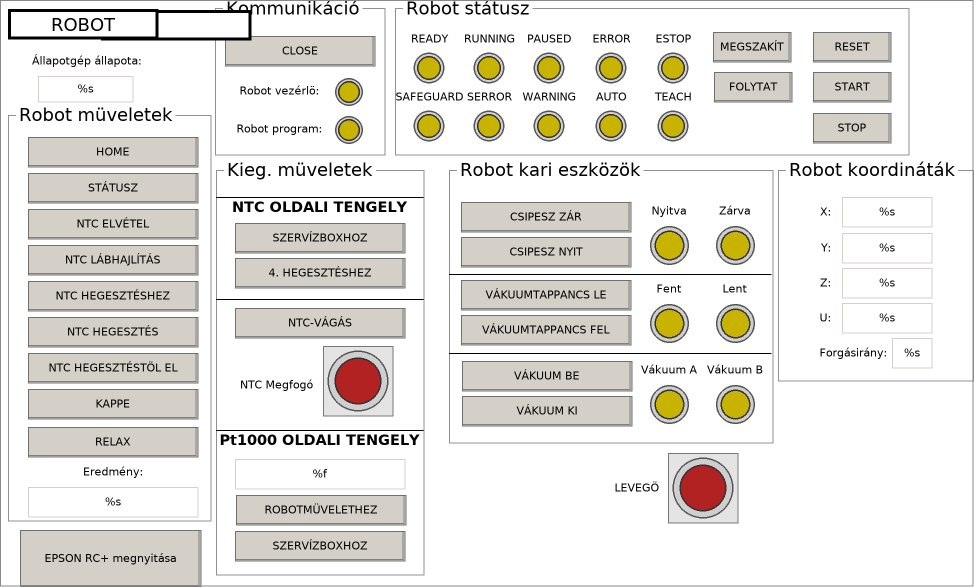
VISUALIZATION Robot  // 974x587
    GroupBox (215,0 170x155), "Kommunikáció"
        Button (10,36 150x30), "OPEN", invisible if: RobotProcess.iState>0, input disabled if: RobotProcess.iState>0
            OnMouseClick: execute { RobotProcess.iState:=1; }
        Button (10,36 150x30), "CLOSE", invisible if: RobotProcess.iState=0, input disabled if: RobotProcess.iState=0
            OnMouseClick: execute { RobotProcess.iState:=200; }
        Lamp1 (116,76 36x32), variable: ROBOTREMOTE.bRobotCommOpen, style: Lamp-Lamp1-Yellow
        Label (23,81 84x20), "Robot vezérlö:"
        Label (9,119 101x20), "Robot program:"
        Lamp1 (116,114 36x32), variable: ROBOTCOMMAND.bRobotCommOpen, style: Lamp-Lamp1-Yellow
    GroupBox (395,0 514x155), "Robot státusz", invisible if: RobotProcess.iState=0, input disabled if: RobotProcess.iState=0
        Lamp1 (16,50 36x36), variable: RobotProcess.baStatus[10], invisible if: ROBOTREMOTE.bRobotCommOpen=FALSE, style: Lamp-Lamp1-Yellow
        Label (6,24 57x30), "READY", invisible if: ROBOTREMOTE.bRobotCommOpen=FALSE
        Lamp1 (76,50 36x36), variable: RobotProcess.baStatus[9], invisible if: ROBOTREMOTE.bRobotCommOpen=FALSE, style: Lamp-Lamp1-Yellow
        Label (66,24 57x30), "RUNNING", invisible if: ROBOTREMOTE.bRobotCommOpen=FALSE
        Lamp1 (136,50 36x36), variable: RobotProcess.baStatus[8], invisible if: ROBOTREMOTE.bRobotCommOpen=FALSE, style: Lamp-Lamp1-Yellow
        Label (126,24 57x30), "PAUSED", invisible if: ROBOTREMOTE.bRobotCommOpen=FALSE
        Lamp1 (198,50 36x36), variable: RobotProcess.baStatus[7], invisible if: ROBOTREMOTE.bRobotCommOpen=FALSE, style: Lamp-Lamp1-Yellow
        Label (188,24 57x30), "ERROR", invisible if: ROBOTREMOTE.bRobotCommOpen=FALSE
        Lamp1 (260,50 36x36), variable: RobotProcess.baStatus[6], invisible if: ROBOTREMOTE.bRobotCommOpen=FALSE, style: Lamp-Lamp1-Yellow
        Label (250,24 57x30), "ESTOP", invisible if: ROBOTREMOTE.bRobotCommOpen=FALSE
        Lamp1 (16,108 36x36), variable: RobotProcess.baStatus[5], invisible if: ROBOTREMOTE.bRobotCommOpen=FALSE, style: Lamp-Lamp1-Yellow
        Label (6,82 57x30), "SAFEGUARD", invisible if: ROBOTREMOTE.bRobotCommOpen=FALSE
        Lamp1 (76,108 36x36), variable: RobotProcess.baStatus[4], invisible if: ROBOTREMOTE.bRobotCommOpen=FALSE, style: Lamp-Lamp1-Yellow
        Label (66,82 57x30), "SERROR", invisible if: ROBOTREMOTE.bRobotCommOpen=FALSE
        Lamp1 (136,108 36x36), variable: RobotProcess.baStatus[3], invisible if: ROBOTREMOTE.bRobotCommOpen=FALSE, style: Lamp-Lamp1-Yellow
        Label (126,82 57x30), "WARNING", invisible if: ROBOTREMOTE.bRobotCommOpen=FALSE
        Lamp1 (198,108 36x36), variable: RobotProcess.baStatus[2], invisible if: ROBOTREMOTE.bRobotCommOpen=FALSE, style: Lamp-Lamp1-Yellow
        Label (188,82 57x30), "AUTO", invisible if: ROBOTREMOTE.bRobotCommOpen=FALSE
        Lamp1 (260,108 36x36), variable: RobotProcess.baStatus[1], invisible if: ROBOTREMOTE.bRobotCommOpen=FALSE, style: Lamp-Lamp1-Yellow
        Label (250,82 57x30), "TEACH", invisible if: ROBOTREMOTE.bRobotCommOpen=FALSE
        RoundedRectangle (-294,10 150x30)
        Button (318,32 78x30), "MEGSZAKÍT"
            OnMouseClick: execute { ROBOTREMOTE.sRobotCommand := 'Pause'; ROBOTREMOTE.bRobotCommandSend := TRUE; }
        Button (319,72 78x30), "FOLYTAT"
            OnMouseClick: execute { ROBOTREMOTE.sRobotCommand := 'Continue'; ROBOTREMOTE.bRobotCommandSend := TRUE; }
        Button (418,32 78x30), "RESET"
            OnMouseClick: execute { ROBOTREMOTE.sRobotCommand := 'Reset'; ROBOTREMOTE.bRobotCommandSend := TRUE; }
        Button (418,72 78x30), "START"
            OnMouseClick: execute {
                ROBOTREMOTE.sRobotCommand := 'Start';
                ROBOTREMOTE.sRobotCommandParam1 := '0';
                ROBOTREMOTE.bRobotCommandSend := TRUE;
            }
        Button (418,113 78x30), "STOP"
            OnMouseClick: execute { ROBOTREMOTE.sRobotCommand := 'Stop'; ROBOTREMOTE.bRobotCommandSend := TRUE; }
    GroupBox (8,107 203x414), "Robot müveletek", invisible if: RobotProcess.iState=0, input disabled if: RobotProcess.iState=0
        Button (20,102 170x30), "NTC ELVÉTEL", invisible if: RobotProcess.iState=0, input disabled if: RobotProcess.iState=0
            OnMouseClick: execute { RobotProcess.s_InRobotTCPCommand := 'NTCHEZ'; }
        Button (20,174 170x30), "NTC HEGESZTÉSHEZ", invisible if: RobotProcess.iState=0, input disabled if: RobotProcess.iState=0
            OnMouseClick: execute { RobotProcess.s_InRobotTCPCommand := 'NTCHEG'; }
        Button (20,246 170x30), "NTC HEGESZTÉSTÖL EL", invisible if: RobotProcess.iState=0, input disabled if: RobotProcess.iState=0
            OnMouseClick: execute { RobotProcess.s_InRobotTCPCommand := 'NTCHEGTOL'; }
        Button (20,282 170x30), "KAPPE", invisible if: RobotProcess.iState=0, input disabled if: RobotProcess.iState=0
            OnMouseClick: execute { RobotProcess.s_InRobotTCPCommand := 'KAPPE'; }
        Button (20,320 170x30), "RELAX", invisible if: RobotProcess.iState=0, input disabled if: RobotProcess.iState=0
            OnMouseClick: execute { RobotProcess.s_InRobotTCPCommand := 'RELAX'; }
        Button (20,30 170x30), "HOME", invisible if: RobotProcess.iState=0, input disabled if: RobotProcess.iState=0
            OnMouseClick: execute { RobotProcess.s_InRobotTCPCommand := 'HOME'; }
        Textfield (20,380 170x30), "%s", text variable: ROBOTCOMMAND.sRobotResult, input disabled if: TRUE
        Label (60,350 90x30), "Eredmény:"
        Button (20,138 170x30), "NTC LÁBHAJLÍTÁS", invisible if: RobotProcess.iState=0, input disabled if: RobotProcess.iState=0
            OnMouseClick: execute { RobotProcess.s_InRobotTCPCommand := 'NTCLAB'; }
        Button (20,66 170x30), "STÁTUSZ", invisible if: RobotProcess.iState=0, input disabled if: RobotProcess.iState=0
            OnMouseClick: execute { RobotProcess.s_InRobotTCPCommand := 'STATUSZ'; }
        Button (20,210 170x30), "NTC HEGESZTÉS", invisible if: RobotProcess.iState=0, input disabled if: RobotProcess.iState=0
            OnMouseClick: execute {
                IF ROBOTCOMMAND.sRobotResult='NTCHEG' THEN
                	RobotProcess.s_InRobotTCPCommand := 'NTCHEG2';
                END_IF
            }
    Textfield (38,76 95x26), "%s", text variable: RobotProcess.iState, input disabled if: TRUE
    GroupBox (216,162 208x413), "Kieg. müveletek", invisible if: RobotProcess.iState=0, input disabled if: RobotProcess.iState=0
        Button (19,146 170x30), "NTC-VÁGÁS", input disabled if: NTCProcess.s_InCommand <> ''
            OnMouseUp: execute {
                IF NTCProcess.s_InCommand = '' THEN
                	NTCProcess.s_InCommand:='VAGAS';
                END_IF
            }
        Button (19,96 170x30), "4. HEGESZTÉSHEZ"
            OnMouseUp: execute { JOZSITENGELY.lrJozsiPosition:=GVL.lrHegesztoPosition4; JOZSITENGELY.sJozsiAxisCommand:='MOVE'; }
        PushSwitch (107,184 70x70), variable: NTCProcess.bMegfogo, behaviour: TOGGLE, style: Switch-PushSwitch-Red
        Label (17,213 87x20), "NTC Megfogó"
        Textfield (19,297 170x30), "%f", text variable: GVL.lrRobotKappePosition
            OnMouseClick: write the text variable via VisuDialogs.Numpad, min -10000, max -1
        Button (19,61 170x30), "SZERVÍZBOXHOZ"
            OnMouseUp: execute { JOZSITENGELY.lrJozsiPosition:=GVL.lrNTCSzervizbox; JOZSITENGELY.sJozsiAxisCommand:='MOVE'; }
        Button (19,369 170x30), "SZERVÍZBOXHOZ"
            OnMouseUp: execute { PISTITENGELY.lrPistiPosition:=GVL.lrPtSzervizbox; PISTITENGELY.sPistiAxisCommand:='MOVE'; }
        Line (0,268) (207,268), "Pt1000 OLDALI TENGELY"
        Line (0,35) (207,35), "NTC OLDALI TENGELY"
        Line (0,137) (207,137)
        Button (20,333 170x30), "ROBOTMÜVELETHEZ"
            OnMouseUp: execute { PISTITENGELY.lrPistiPosition:=GVL.lrRobotKappePosition; PISTITENGELY.sPistiAxisCommand:='MOVE'; }
    Label (27,46 120x30), "Állapotgép állapota:"
    RoundedRectangle (8,9 150x30)
    Label (8,10 150x30), "ROBOT"
    GroupBox (449,162 324x281), "Robot kari eszközök", invisible if: RobotProcess.iState=0, input disabled if: RobotProcess.iState=0
        Button (12,40 170x30), "CSIPESZ ZÁR", invisible if: RobotProcess.iState=0, input disabled if: RobotProcess.iState=0
            OnMouseClick: execute { RobotProcess.s_InRobotTCPCommand := 'CSIPESZ_ZAR'; }
        Button (12,75 170x30), "CSIPESZ NYIT", invisible if: RobotProcess.iState=0, input disabled if: RobotProcess.iState=0
            OnMouseClick: execute { RobotProcess.s_InRobotTCPCommand := 'CSIPESZ_NYIT'; }
        Group (12,118 170x65)
            Button (0,0 170x30), "VÁKUUMTAPPANCS LE", invisible if: RobotProcess.iState=0, input disabled if: RobotProcess.iState=0
                OnMouseClick: execute { RobotProcess.s_InRobotTCPCommand := 'SZIPPANTO_LE'; }
            Button (0,35 170x30), "VÁKUUMTAPPANCS FEL", invisible if: RobotProcess.iState=0, input disabled if: RobotProcess.iState=0
                OnMouseClick: execute { RobotProcess.s_InRobotTCPCommand := 'SZIPPANTO_FEL'; }
        Group (13,199 170x65)
            Button (0,35 170x30), "VÁKUUM KI", invisible if: RobotProcess.iState=0, input disabled if: RobotProcess.iState=0
                OnMouseClick: execute { RobotProcess.s_InRobotTCPCommand := 'VAKUUM_KI'; }
            Button (0,0 170x30), "VÁKUUM BE", invisible if: RobotProcess.iState=0, input disabled if: RobotProcess.iState=0
                OnMouseClick: execute { RobotProcess.s_InRobotTCPCommand := 'VAKUUM_BE'; }
        Lamp1 (198,61 45x45), variable: GVL.stRobotStatusz.bCsipeszNyitva, style: Lamp-Lamp1-Yellow
        Label (190,39 60x20), "Nyitva"
        Lamp1 (264,61 45x45), variable: GVL.stRobotStatusz.bCsipeszZarva, style: Lamp-Lamp1-Yellow
        Label (256,39 60x20), "Zárva"
        Lamp1 (198,139 45x45), variable: GVL.stRobotStatusz.bVakuumSzippantoFent, style: Lamp-Lamp1-Yellow
        Label (190,117 60x20), "Fent"
        Lamp1 (264,139 45x45), variable: GVL.stRobotStatusz.bVakuumSzippantoLent, style: Lamp-Lamp1-Yellow
        Label (256,117 60x20), "Lent"
        Lamp1 (198,220 45x45), variable: GVL.stRobotStatusz.bVakuumA, style: Lamp-Lamp1-Yellow
        Label (190,198 60x20), "Vákuum A"
        Lamp1 (264,220 45x45), variable: GVL.stRobotStatusz.bVakuumB, style: Lamp-Lamp1-Yellow
        Label (256,198 60x20), "Vákuum B"
        Line (0,112) (322,112)
        Line (0,191) (322,191)
    GroupBox (778,162 196x219), "Robot koordináták", invisible if: RobotProcess.iState=0, input disabled if: RobotProcess.iState=0
        Group (36,35 118x171)
            Label (0,5 20x20), "X:"
            Textfield (28,0 90x30), "%s", text variable: GVL.stRobotStatusz.rX
            Label (0,41 20x20), "Y:"
            Textfield (28,36 90x30), "%s", text variable: GVL.stRobotStatusz.rY
            Label (0,76 20x20), "Z:"
            Textfield (28,71 90x30), "%s", text variable: GVL.stRobotStatusz.rZ
            Textfield (28,106 90x30), "%s", text variable: GVL.stRobotStatusz.rU
            Label (0,111 20x20), "U:"
            Textfield (78,141 40x30), "%s", text variable: GVL.stRobotStatusz.sHand
            Label (0,146 76x20), "Forgásirány:"
    Group (607,453 131x70), invisible if: RobotProcess.iState=0, input disabled if: RobotProcess.iState=0
        PushSwitch (61,0 70x70), variable: MAIN.bLevego, behaviour: TOGGLE, style: Switch-PushSwitch-Red
        Label (0,20 55x30), "LEVEGÖ"
    Button (20,530 181x57), "EPSON RC+ megnyitása"
        OnMouseUp: ExecuteCommand ExecuteCommand=ExecuteCommand=[Command=ExecuteClientProgram, Value='C:\EpsonRC70\exe\erc70.exe']
END_VISUALIZATION

(* stored: Version 1.1.0.1, ProductVersion 3.1.4024.11
   Visu Robot: Id {2fff07b8-4fc5-4075-b558-515cbd3f308c} *)
